Staubli VAL3: EnterPageKey.pgx

program EnterPageKey(num& x_nKey, num& x_nSelect, string& x_sItem)
  local string l_sStr
  local num l_nKey
  local string l_sEmpty
  local string l_sValue
  local num l_nItem
  local num l_nView
  local string l_sItem
  local point lp
  local string l_sYN[2]
  local bool l_bRes
  local num l_nTemp
  local num l_i
begin
  //
  //编辑项目
  switch x_nSelect
    //
    case 0

    break
    //砂带补偿量
    default
      if x_nKey==270
        call user:editNum(x_sItem,sListItemValue[x_nSelect],l_nTemp,x_nSelect)
        if l_nTemp>0.08
          popUpMsg("最大0.08")
          l_nTemp=0.08
          sParameter[x_nSelect]=sPath[x_nSelect-1]
          sListItemValue[0]=toString(".4",PublicData:nDelta)
          call user:strlength(sParameter[l_i],user:nBottomX/2)
          l_sValue=sListItemValue[l_i]
          call user:strlength(l_sValue,user:nBottomX/2+1)
          sParameter[l_i]=sParameter[l_i]+":"+l_sValue
        endIf

        if prd:libLoad("Disk://Traj/"+sPath[x_nSelect-1])==0
          prd:nCompDelta=l_nTemp
          prd:libSave()
        endIf
      endIf

    break
  endSwitch
  if x_nKey==270
    bUserRefresh=true
    bListRefresh=true
  endIf
end
